// TIA Portal V18 export
// export: Created 2026-06-12T00:00:00Z, ExportSetting WithDefaults, DisplayName Totally Integrated Automation Portal, DisplayVersion V18
TagTable "HMI_Tags"
  AI_LT3203_PV : Real  (PLC tag AI_LT3203_PV, HMI_Connection_1, 1 s)
  AI_TT3204_PV : Real  (PLC tag AI_TT3204_PV, HMI_Connection_1, 1 s)
  AI_LT3209_PV : Real  (PLC tag AI_LT3209_PV, HMI_Connection_1, 1 s)
  AI_TT3208_PV : Real  (PLC tag AI_TT3208_PV, HMI_Connection_1, 1 s)
  AI_LT3213_PV : Real  (PLC tag AI_LT3213_PV, HMI_Connection_1, 1 s)
  AI_TT3214_PV : Real  (PLC tag AI_TT3214_PV, HMI_Connection_1, 1 s)
  AI_LT3218_PV : Real  (PLC tag AI_LT3218_PV, HMI_Connection_1, 1 s)
  AI_TT3219_PV : Real  (PLC tag AI_TT3219_PV, HMI_Connection_1, 1 s)
  AI_BON1_Chay : Bool  (PLC tag AI_BON1_Chay, HMI_Connection_1, 1 s)
  AI_BON2_Chay : Bool  (PLC tag AI_BON2_Chay, HMI_Connection_1, 1 s)
  AI_BON3_Chay : Bool  (PLC tag AI_BON3_Chay, HMI_Connection_1, 1 s)
  AI_BON4_Chay : Bool  (PLC tag AI_BON4_Chay, HMI_Connection_1, 1 s)
  AI_PUMP3264_Chay : Bool  (PLC tag AI_PUMP3264_Chay, HMI_Connection_1, 1 s)
  AI_PUMP3265_Chay : Bool  (PLC tag AI_PUMP3265_Chay, HMI_Connection_1, 1 s)
  AI_Logged_In : Int  (PLC tag AI_Logged_In, HMI_Connection_1, 1 s)
